{attribute 'qualified_only'}
{attribute 'strict'}
{attribute 'to_string'}
TYPE E_TransferCapability :
(
	Unknown := 0,
	SendOnly,
	ReveiveOnly,
	Bidirectional
);
END_TYPE

(* stored: Version 1.1.0.1, ProductVersion 3.1.4026.18
   DUT E_TransferCapability: Id {3813247c-1b3d-4799-ac2b-52e0e372a97c} *)
